FUNCTION_BLOCK fbPassManager
VAR_INPUT
	sUserToChange		: WSTRING;
END_VAR
VAR_OUTPUT
END_VAR
VAR
	
	nYear				: REAL;
	nMonth				: REAL;
	bInitOK 			: BOOL := FALSE;
	wsNewPass			: WSTRING(255);
	wsOldPass			: WSTRING(255);
	bChangePass			: BOOL;
	
END_VAR
VAR PERSISTENT 
	
	nYear_per				: REAL;
	nMonth_per				: REAL;	
	
END_VAR

ChangePass();

METHOD ChangePass : BOOL
VAR_INST
	bTimeEnd		: BOOL;
	tonTimeEnd		: TON;
END_VAR
IF NOT bTimeEnd THEN
	IF THIS^.GetTime()  = 2 THEN
		IF THIS^.SetPass() THEN
			tonTimeEnd( IN := FALSE, PT := T#1M);
			bTimeEnd   := TRUE;
			ChangePass := TRUE;
		END_IF
	ELSE
		IF THIS^.GetTime()  = 1 THEN
			tonTimeEnd( IN := FALSE, PT := T#1M);
			bTimeEnd   := TRUE;			
		END_IF
	END_IF
ELSE
	tonTimeEnd( IN := TRUE, PT := T#1M);
	IF tonTimeEnd.Q THEN
		bTimeEnd := FALSE;
	END_IF
	ChangePass := FALSE;
END_IF
END_METHOD

METHOD GeneratingPass : WSTRING
VAR_INPUT
	nMonth : REAL;
	nYear  : REAL;
END_VAR
VAR_INST
		lnPass				: LREAL;
		lnPass_				: DINT;

		fbFormat			: FB_FormatString;
		sNewPass			: STRING(255);
		uiLicznik 			: UINT;
		wsNewPass_			: WSTRING(255);
END_VAR

lnPass := (EXPT(nMonth,4) + 5*nYear) - ( nYear - 1950)* EXPT(( nMonth - 3 ), 3) + ( EXPT( nMonth - 4, 2)*(nYear - 2040) * (nMonth -1))  + 50000;
lnPass_ := LREAL_TO_DINT(lnPass);
fbFormat( sFormat := '%d', arg1 := F_DINT(lnPass_), sOut => sNewPass);
FOR uiLicznik :=0 TO 255 DO
	wsNewPass_[uiLicznik] := sNewPass[uiLicznik];
END_FOR
GeneratingPass := wsNewPass_;
END_METHOD

METHOD GetTime : UINT
VAR_INPUT
END_VAR
VAR_INST
	fbGetTime	: NT_GetTime;
	bStart		: BOOL;
	nStan		: UINT := 0;
END_VAR
IF NOT bStart THEN
	bStart 	:= TRUE;
	nStan  	:= 10;
	GetTime := 0;
ELSE
	CASE nStan OF 
		0:
			fbGetTime( NETID := '', Start := FALSE);
			GetTime := 0;
		10 :
			fbGetTime( NETID := '', Start := TRUE);
			GetTime := 0;
			IF NOT fbGetTime.BUSY THEN
				nStan  := 20;
			END_IF	
		
		20 :
			nYear   := WORD_TO_UINT(fbGetTime.TIMESTR.wYear);
			nMonth  := WORD_TO_UINT(fbGetTime.TIMESTR.wMonth);
			nStan   := 0;
			bStart  := FALSE;
			IF nYear = nYear_per AND nMonth = nMonth_per THEN
				GetTime := 1;
			ELSE
				nYear_per := nYear;
				nMonth_per  := nMonth;
				GetTime := 2;
			END_IF
			
	END_CASE
END_IF
END_METHOD

METHOD SetPass : BOOL
VAR_INPUT
END_VAR
VAR_INST
	pClient				: POINTER TO VisuElems.VisuStructClientData; 
	fbVisuUserMgmt		: VisuUserManagement.VisuUserMgmt;
	dwUserDB			: DWORD;
END_VAR
wsNewPass := THIS^.GeneratingPass( nMonth := nMonth ,nYear := nYear ) ;
fbVisuUserMgmt();
dwUserDB := fbVisuUserMgmt.GetUserDBAsCopy();
fbVisuUserMgmt.ChangeUserPassword(dwUserDB,sUserToChange, wsNewPass, "");
fbVisuUserMgmt.SetNewUserDB( dwUserDB := dwUserDB,bResultOK := TRUE);
SetPass := TRUE;
END_METHOD

END_FUNCTION_BLOCK

(* stored: Version 1.1.0.1, ProductVersion 3.1.4024.15
   POU fbPassManager: Id {d89b5525-1a7c-4642-9959-f13aebd7546e}, SpecialFunc None
   Method ChangePass: Id {b0cb95e6-7ea9-4abd-8e70-ad46e58cedb6}
   Method GeneratingPass: Id {012e5846-3956-4428-b8e0-e22df266645a}
   Method GetTime: Id {639d54ad-dc2b-4551-a06e-5e1513e5c6b5}
   Method SetPass: Id {6e3823e8-2576-4f7d-a196-b2e6cf5d9823} *)
